// TIA Portal V17 export
// export: Created 2025-06-26T06:49:13.299935Z, ExportSetting WithDefaults, DisplayName Totally Integrated Automation Portal, DisplayVersion V17 Update 8, DisplayName TIA Portal Openness, DisplayVersion V17 Update 8, DisplayName TIA Portal Version Control Interface, DisplayVersion V17, DisplayName STEP 7 Professional, DisplayVersion V17 Update 8, DisplayName STEP 7 Safety, DisplayVersion V17 Update 6, DisplayName WinCC Advanced, DisplayVersion V17 Update 8
FUNCTION_BLOCK "fbOilRecovery"   // FB58, FBD
TITLE = Run once every X times with a fixed valve setpoint
{ S7_Optimized_Access := 'TRUE' }
AUTHOR : Heaten
VERSION : 0.1
// stored: AutoNumber true, IsIECCheckEnabled false, IsRetainMemResEnabled false, MemoryReserve 0, SetENOAutomatically false, UDAEnableTagReadback false
   VAR_INPUT
      bEnable : Bool;
      bReset : Bool;
   END_VAR
   VAR_OUTPUT
      bOut : Bool;
      fOut : Real;
   END_VAR
   VAR_IN_OUT
      sTag : "stOilRecovery";
   END_VAR
   VAR
      Controller : "fbOneShotRegulator";
      epEnabled : R_TRIG;
      RunCounter { S7_SetPoint := 'True'} : UInt;
      RunCounterMod : UInt;
   END_VAR
   VAR RETAIN
      Count { S7_SetPoint := 'True'} : Bool;
   END_VAR
   VAR_TEMP
      bEnabled : Bool;
   END_VAR
BEGIN

REGION Network 1: Run signal
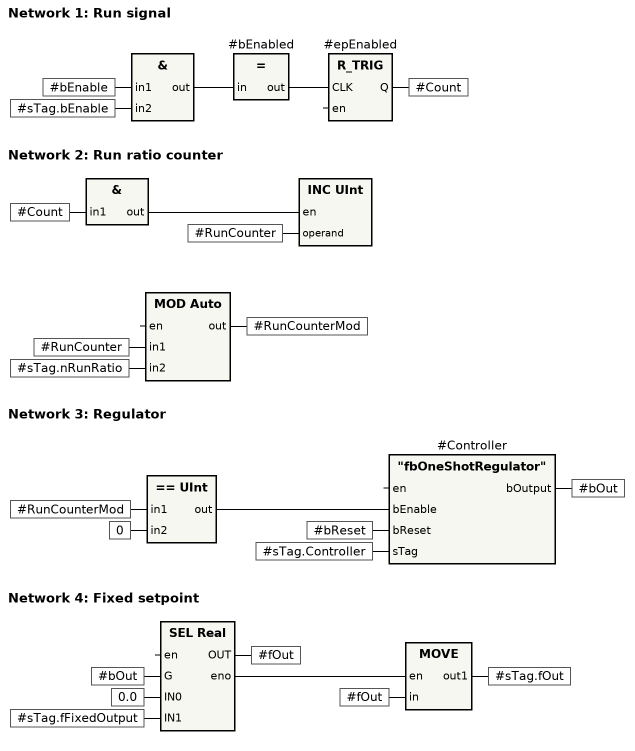
   #bEnabled := #bEnable AND #sTag.bEnable;
   #epEnabled(CLK := #bEnabled, Q => #Count);   // R_TRIG
END_REGION

REGION Network 2: Run ratio counter
   IF #Count THEN #RunCounter := #RunCounter + 1; END_IF;
   #RunCounterMod := #RunCounter MOD #sTag.nRunRatio;
END_REGION

REGION Network 3: Regulator
   // RunCounterMod is 0 every nth count.
   #Controller(bEnable := #RunCounterMod = 0, bReset := #bReset, sTag := #sTag.Controller, bOutput => #bOut);   // "fbOneShotRegulator"
END_REGION

REGION Network 4: Fixed setpoint
   // ENO of a box is taken as its EN; it also drops when the box reports an error
   #fOut := SEL(G := #bOut, IN0 := 0.0, IN1 := #sTag.fFixedOutput);
   #sTag.fOut := #fOut;
END_REGION
END_FUNCTION_BLOCK
